KUKA KRL data list: data.dat

&ACCESS RVO
DEFDAT test_data
  ; KRL Data file example

  ; Global constants
  DECL GLOBAL CONST INT MAX_SPEED = 100
  DECL GLOBAL CONST REAL PI = 3.14159

  ; Global variables
  DECL GLOBAL INT counter
  DECL GLOBAL BOOL emergency_stop

  ; Position data
  DECL GLOBAL E6POS home_pos = {X 0.0, Y 0.0, Z 800.0, A 0.0, B 0.0, C 0.0, S 2, T 10}
  DECL GLOBAL E6POS work_pos[10]

  ; Frame data
  DECL GLOBAL FRAME tool_offset = {X 0.0, Y 0.0, Z 150.0, A 0.0, B 0.0, C 0.0}
  DECL GLOBAL FRAME base_frame = {X 0.0, Y 0.0, Z 0.0, A 0.0, B 0.0, C 0.0}

  ; Tool data
  DECL GLOBAL TOOL_DATA gripper = {X 0.0, Y 0.0, Z 200.0, A 0.0, B 0.0, C 0.0}

  ; Load data
  DECL GLOBAL LOAD_DATA payload = {M 5.0, CM {X 0.0, Y 0.0, Z 50.0, A 0.0, B 0.0, C 0.0}, J {X 0.0, Y 0.0, Z 0.0}}

ENDDAT
